(* PLC project  *)

CONFIGURATION FSOE_Slot_1
END_CONFIGURATION
